{attribute 'GeneratedUsingTerminal: EK1100-0000-0018'}
{attribute addProperty BoxType "EK1100-0000-0018"}
{attribute addProperty Id "Beckhoff_ER3xxxEK1122Beckhoff_ER3xxxEK1122_6C0C5CDA618"}
{attribute addProperty CRC "4038188257"}
{attribute addProperty Size "618"}
TYPE Beckhoff_ER3xxx_F0B1DCE1 EXTENDS EK1100_1FC0878B :
STRUCT
	{attribute addProperty Name "Beckhoff_ER3xxxEK1122"}
	{attribute addProperty PreviousPort "Beckhoff ER3xxx : B"}
	Beckhoff_ER3xxxEK1122 : Beckhoff_ER3xxxEK1122_6C0C5CDA;
END_STRUCT
END_TYPE

(* stored: Version 1.2.0.0, ProductVersion 3.1.4024.9
   DUT Beckhoff_ER3xxx_F0B1DCE1: Id {ca994823-7386-47ef-9829-ef791d2ab8a5} *)
